TYPE ST_DOS_Diagnosis :
STRUCT
	Chanel_0	: ST_DOS_Chanel_Diagnosis;
	Chanel_1	: ST_DOS_Chanel_Diagnosis;
	Chanel_2	: ST_DOS_Chanel_Diagnosis;
	Chanel_3	: ST_DOS_Chanel_Diagnosis;
	Chanel_4	: ST_DOS_Chanel_Diagnosis;
	Chanel_5	: ST_DOS_Chanel_Diagnosis;
	Chanel_6	: ST_DOS_Chanel_Diagnosis;
	Chanel_7	: ST_DOS_Chanel_Diagnosis;
END_STRUCT
END_TYPE

(* stored: Version 1.1.0.1
   DUT ST_DOS_Diagnosis: Id {94e8c0cf-39ac-4aa9-a360-1c5d267cb018} *)
